{attribute 'hide_all_locals'}
FUNCTION_BLOCK FB_1_ROB EXTENDS FB_0_Base 
// IMPLEMENTS ITF_1_Robot

VAR_INPUT
	SET_R: stSettings_Rob;
	PM: FB_PointManager;
	COMM: POINTER TO FB_1_COMM := ADR(emptyCOMM);

END_VAR


VAR_OUTPUT
	HMI_ROB: stHMI_ROB;

	nCommandID: UINT;
	eCommandStatus: eProgress;
	eCommandResult: eResult := NONE;
	
	TCPPos_PLCUnit : ST_Pose;				// mm/rad
	JointPos_PLCUnit: stJoint6;			//rad
	JointVel_PLCUnit: stJoint6;
    TCPVel_PLCUnit : ST_Pose;
END_VAR

VAR
    T_W_B      : ST_TransformMatrix;		//Set in fb_Init
	index: INT;
	
	//BAHANDLER
	Idcounter: UINT:=1000;


	
	_INIT_ROB: BOOL;
	_Homed: BOOL;
  _cancelRequestID : UINT;
  _cancelNotificationSent : BOOL;
  _lifecycleStopRequested : BOOL;
  _lifecycleStopComplete : BOOL;
END_VAR

{warning 'Add property implementation'}
PROPERTY ActualJointPosition : stJoint6
GET
ActualJointPosition := JointPos_PLCUnit;
END_GET
SET
JointPos_PLCUnit:= ActualJointPosition;
END_SET
END_PROPERTY

{warning 'Add property implementation'}
  PROPERTY ActualJointVelocity : stJoint6
GET
ActualJointVelocity := JointVel_PLCUnit;
END_GET
SET
JointVel_PLCUnit := ActualJointVelocity;
END_SET
END_PROPERTY

{warning 'Add property implementation'}
  PROPERTY ActualPosition : ST_Pose
GET
ActualPosition := TCPPos_PLCUnit;
END_GET
SET
TCPPos_PLCUnit:= ActualPosition;
END_SET
END_PROPERTY

{warning 'Add property implementation'}
 PROPERTY ActualVelocity : ST_Pose
GET
ActualVelocity := TCPVel_PLCUnit;
END_GET
SET
TCPVel_PLCUnit:= ActualVelocity;
END_SET
END_PROPERTY

METHOD PROTECTED AllocateCommandID : UINT
IF Idcounter >= 65534 THEN
  Idcounter := 1001;
ELSE
	Idcounter := Idcounter + 1;
END_IF

AllocateCommandID := Idcounter;
END_METHOD

PROPERTY CanAcceptCommand : BOOL
GET
CanAcceptCommand :=
    (State = eState.Active)
    AND NOT RecoveryPending
    AND NOT ((nCommandID <> 0)
      AND ((eCommandStatus = INIT)
        OR (eCommandStatus = ACKNOWLEDGE)
        OR (eCommandStatus = RUNNING)));

IF CanAcceptCommand AND (COMM <> 0) AND (COMM <> ADR(emptyCOMM)) THEN
    CanAcceptCommand := COMM^.CanAcceptCommand;
END_IF
END_GET
END_PROPERTY

{warning 'Override with your own Method in final FB'}
METHOD CommandHandler : UINT
VAR_INPUT
    Cmd      : eCommands;
    Settings : stCommand_Settings := SETUP.emptySettings;
END_VAR

VAR

	CancelRes: BOOL;
END_VAR
(* Base implementation: unsupported. Final robot FB overrides this method. *)
CommandHandler := 0;
END_METHOD

PROPERTY CommandID : UINT
GET
CommandID := nCommandID;
END_GET
SET
 nCommandID := CommandID;
END_SET
END_PROPERTY

PROPERTY CommandResult : eResult
GET
CommandResult := COMM^.CommandResult;
END_GET
SET
eCommandResult := CommandResult;
IF (COMM <> 0) AND (COMM <> ADR(emptyCOMM)) THEN
    COMM^.CommandResult := CommandResult;
END_IF
END_SET
END_PROPERTY

PROPERTY CommandState : eProgress
GET
CommandState := COMM^.CommandState;
END_GET
SET
eCommandStatus := CommandState;
IF (COMM <> 0) AND (COMM <> ADR(emptyCOMM)) THEN
    COMM^.CommandState := CommandState;
END_IF
END_SET
END_PROPERTY

ACTION CYCLIC_ROB:
IF NOT _INIT_ROB THEN
	_INIT_ROB:=TRUE;
	SETUP_ROB();
END_IF

CYCLIC_BASE();
PM.HMI_PM.xCurrentTcp := ActualPosition;
PM(pRobot := THIS);

IF (State <> eState.Deactivating)
   AND (State <> eState.ErrorProcessing)
   AND (State <> eState.ShuttingDown) THEN
  _lifecycleStopRequested := FALSE;
  _lifecycleStopComplete := FALSE;
END_IF


// HMI display mirrors: _tcppos/_jointpos stay in PLC standard (mm/rad); display in mm/deg.
HMI_ROB.TCPPos_HMIUnit := ChangePoseToHMIStandard(Pose := TCPPos_PLCUnit);

HMI_ROB.JointPos_HMIUnit.joint1 := ChangeRealToHMIStandard(
    Value := JointPos_PLCUnit.joint1, Category := eUnitCategory.Joint);
HMI_ROB.JointPos_HMIUnit.joint2 := ChangeRealToHMIStandard(
    Value := JointPos_PLCUnit.joint2, Category := eUnitCategory.Joint);
HMI_ROB.JointPos_HMIUnit.joint3 := ChangeRealToHMIStandard(
    Value := JointPos_PLCUnit.joint3, Category := eUnitCategory.Joint);
HMI_ROB.JointPos_HMIUnit.joint4 := ChangeRealToHMIStandard(
    Value := JointPos_PLCUnit.joint4, Category := eUnitCategory.Joint);
HMI_ROB.JointPos_HMIUnit.joint5 := ChangeRealToHMIStandard(
    Value := JointPos_PLCUnit.joint5, Category := eUnitCategory.Joint);
HMI_ROB.JointPos_HMIUnit.joint6 := ChangeRealToHMIStandard(
    Value := JointPos_PLCUnit.joint6, Category := eUnitCategory.Joint);

// Adopt communication faults + health so the robot reflects its comm child.
IF COMM <> 0 AND COMM <> ADR(emptyCOMM) THEN
  COMM^.MESSENGER.ParentMessenger := ADR(MESSENGER);
	IF COMM^.State = eState.ErrorProcessing OR COMM^.MESSENGER.HasActivError THEN
        SetRecoveryMode(Mode := COMM^.RecoveryMode);
		Messenger.AddError(eMessageCategories.ParentFailed,Path,'Communication module in error');
	END_IF
END_IF




FOR index := TO_INT(LOWER_BOUND(Skills, 1)) TO TO_INT(UPPER_BOUND(Skills, 1)) DO
    IF Skills[index] <> 0 THEN
        Skills[index]^.CYCLIC_SKILL();
    END_IF
END_FOR






// --------------PROPS------------

//ActualJointPosition: DONE
//ActualJointVelocity DONE
//ActualTCPPosition: DONE
//ActualTCPVelocity: DONE
//InCollision: depend on Robot Type //TODO
//Mode: depend on RobotType	//TODO

//RobotMoving:
HMI_ROB.bMoving :=
  (ABS(TCPVel_PLCUnit.X)  > SET_R.LinearStandStillLimit) OR
  (ABS(TCPVel_PLCUnit.Y)  > SET_R.LinearStandStillLimit) OR
  (ABS(TCPVel_PLCUnit.Z)  > SET_R.LinearStandStillLimit) OR
  (ABS(TCPVel_PLCUnit.roll) > SET_R.AngularStandStillLimit) OR
  (ABS(TCPVel_PLCUnit.pitch) > SET_R.AngularStandStillLimit) OR
  (ABS(TCPVel_PLCUnit.yaw) > SET_R.AngularStandStillLimit);
	
// Generic robot command contributes to FB_0_Base.Busy. Terminal command values remain latched,
// therefore only non-terminal phases make the robot busy.
HMI_BASE.bBusy := (nCommandID <> 0)
  AND ((eCommandStatus = INIT)
    OR (eCommandStatus = ACKNOWLEDGE)
    OR (eCommandStatus = RUNNING));

IF (COMM <> 0) AND (COMM <> ADR(emptyCOMM)) THEN
  HMI_BASE.bBusy := HMI_BASE.bBusy OR COMM^.StopPending;
END_IF

// Ready means: the robot can accept a NEW semantic command now.
HMI_ROB.bOperational := Operational;
END_ACTION

METHOD PROTECTED EnsureMotionStopped : BOOL
EnsureMotionStopped := FALSE;

    IF (COMM = 0) OR (COMM = ADR(emptyCOMM)) THEN
      EnsureMotionStopped := TRUE;
      RETURN;
    END_IF

    IF NOT _lifecycleStopRequested THEN
      IF NOT COMM^.StopMotion() THEN
        Messenger.AddError(
          eMessageCategories.HardwareFailure,
          CONCAT(Path, '.StopMotion'),
          'Communication adapter rejected the lifecycle stop request');
        RETURN;
      END_IF
      _lifecycleStopRequested := TRUE;
    END_IF

    IF COMM^.MotionStopped THEN
      _lifecycleStopComplete := TRUE;
    END_IF

    EnsureMotionStopped := _lifecycleStopComplete;
END_METHOD

METHOD FB_Init : BOOL
  VAR_INPUT
    bInitRetains : BOOL;
    bInCopyCode : BOOL;
  END_VAR
  VAR
    iRobot : UINT;
  END_VAR
SUPER^.FB_Init(bInitRetains := bInitRetains, bInCopyCode := bInCopyCode);


T_W_B := FromPose(SET_R.InstallationPose);





IF SETUP.nRobCount < SETUP.MaxNrofRobots THEN
	SETUP.nRobCount := SETUP.nRobCount + 1;
	SETUP.apRobot[SETUP.nRobCount+1] := THIS;
	FB_Init := TRUE;
END_IF
END_METHOD

PROPERTY Homed : BOOL
GET
Homed:=_Homed;
END_GET
SET
_Homed:=Homed;
END_SET
END_PROPERTY

{warning 'Add method implementation '}
METHOD Homing : UINT


VAR
	Config: stCommand_Settings;
END_VAR

Config.Velocity := SET_R.HomingVelocity;

Homing:= CommandHandler(Cmd:=eCommands.Homing,Settings:=Config);
END_METHOD

PROPERTY InSavePosition : BOOL
GET
VAR
    joints : stJoint6;
END_VAR
joints := ActualJointPosition;

InSavePosition :=
    (ABS(joints.joint1 - SET_R.ManualSecurePosition.joint1) <= SET_R.SafePositionTolerance) AND
    (ABS(joints.joint2 - SET_R.ManualSecurePosition.joint2) <= SET_R.SafePositionTolerance) AND
    (ABS(joints.joint3 - SET_R.ManualSecurePosition.joint3) <= SET_R.SafePositionTolerance) AND
    (ABS(joints.joint4 - SET_R.ManualSecurePosition.joint4) <= SET_R.SafePositionTolerance) AND
    (ABS(joints.joint5 - SET_R.ManualSecurePosition.joint5) <= SET_R.SafePositionTolerance) AND
    (ABS(joints.joint6 - SET_R.ManualSecurePosition.joint6) <= SET_R.SafePositionTolerance);
END_GET
END_PROPERTY

{warning 'OVERRIDE'}
PROPERTY IsInCollision : BOOL
GET
IsInCollision := HMI_ROB.bInCollision;
END_GET
END_PROPERTY

PROPERTY IsMoving : BOOL
GET
IsMoving := HMI_ROB.bMoving;
END_GET
SET
HMI_ROB.bMoving := IsMoving;
END_SET
END_PROPERTY

METHOD MoveToHomePosition : UINT

VAR
    settings : stCommand_Settings;
END_VAR
MoveToHomePosition := 0;
settings.Velocity := SET_R.HomingVelocity;

IF PM.Load(SET_R.NameOfHomePosition) = SUCCESS THEN
    settings.Pose := PM.LoadedPose;
    MoveToHomePosition := CommandHandler(Cmd := eCommands.MoveJ, Settings := settings);
ELSE
    Messenger.AddError(eMessageCategories.MissingData, Path, 'Home Position not found, aborted');
END_IF
END_METHOD

METHOD MoveToSafePosition : UINT

VAR
    settings : stCommand_Settings;
END_VAR
settings.Velocity := SET_R.HomingVelocity;

IF SET_R.UseSavedSecurePosition THEN							//Not made: Able to save a Saveposition		
	IF PM.Load(SET_R.NameOfSavedSecurePosition) = SUCCESS THEN												
		settings.Pose := PM.LoadedPose;
		MoveToSafePosition := CommandHandler(Cmd := eCommands.MoveJ, Settings := settings);
		RETURN;
	ELSE
		Messenger.AddWarn(eMessageCategories.MissingData,Path,'Secure Position not found, using Manual Position');
		
	END_IF
END_IF


settings.Joints := SET_R.ManualSecurePosition;
MoveToSafePosition := CommandHandler(Cmd := eCommands.MoveJJoints, Settings := settings);
END_METHOD

METHOD PROTECTED OnActivate : eResult
VAR_INPUT
END_VAR

VAR
	eParentResult: eResult;
	myResult: ERESULT;
END_VAR

VAR //YOUR CODE
	succ : BOOL;
END_VAR
eParentResult := SUPER^.OnActivate();
//--------------------------------------------------
myResult:=NONE;
// ----- YOUR CODE HERE (incl. Alarms) -------------

IF Comm^.LastTransitionType = eTransitions.Activate THEN
	IF Comm^.LastTransitionResult = SUCCESS THEN
		myResult:=SUCCESS;
	END_IF
ELSE
	COMM^.Activate();
END_IF

IF SIMMODE THEN
		myResult:=SUCCESS;
END_IF

// ----- END YOUR CODE -----------------------------
//--------------------------------------------------
OnActivate := CombineResults(eParentResult,myResult);
END_METHOD

METHOD PROTECTED OnCleanup : eResult
VAR_INPUT
END_VAR

VAR
	eParentResult: eResult;
	myResult: ERESULT;
END_VAR

VAR //YOUR CODE
	succ : BOOL;
END_VAR
eParentResult := SUPER^.OnCleanup();
//--------------------------------------------------
myResult:=NONE;
// ----- YOUR CODE HERE (incl. Alarms) -------------

IF Comm^.LastTransitionType = eTransitions.Cleanup THEN
	IF Comm^.LastTransitionResult = SUCCESS THEN
		myResult:=SUCCESS;
	END_IF
ELSE
	COMM^.Cleanup();
END_IF

// ----- END YOUR CODE -----------------------------
//--------------------------------------------------
OnCleanup := CombineResults(eParentResult,myResult);
END_METHOD

METHOD PROTECTED OnConfigure : eResult
VAR_INPUT
END_VAR

VAR
	eParentResult: eResult;
	myResult: ERESULT;
END_VAR

VAR //YOUR CODE
	succ : BOOL;
END_VAR
eParentResult := SUPER^.OnConfigure();
//--------------------------------------------------
myResult:=NONE;
// ----- YOUR CODE HERE (incl. Alarms) -------------


IF Comm^.LastTransitionType = eTransitions.Configure THEN
	
	IF Comm^.LastTransitionResult = SUCCESS AND COMM^.Connected  THEN
		myResult:=SUCCESS;
	END_IF
ELSE
	COMM^.Configure();
END_IF

IF SIMMODE THEN
		myResult:=SUCCESS;
END_IF



IF NOT PM.Initialise(sName := Name) = SUCCESS THEN
	myResult:=NONE;
END_IF

PM.LoadAllFromFile();

// ----- END YOUR CODE -----------------------------
//--------------------------------------------------
OnConfigure := CombineResults(eParentResult,myResult);
END_METHOD

METHOD PROTECTED OnDeactivate : eResult
VAR_INPUT
END_VAR

VAR
	eParentResult: eResult;
	myResult: ERESULT;
END_VAR

VAR //YOUR CODE
	succ : BOOL;
END_VAR
eParentResult := SUPER^.OnDeactivate();

IF NOT EnsureMotionStopped() THEN
  OnDeactivate := CombineResults(eParentResult, eResult.NONE);
  RETURN;
END_IF
//--------------------------------------------------
myResult:=NONE;
// ----- YOUR CODE HERE (incl. Alarms) -------------

IF Comm^.LastTransitionType = eTransitions.Deactivate THEN
	IF Comm^.LastTransitionResult = SUCCESS THEN
		myResult:=SUCCESS;
	END_IF
ELSE
	COMM^.Deactivate();
END_IF

// ----- END YOUR CODE -----------------------------
//--------------------------------------------------
OnDeactivate := CombineResults(eParentResult,myResult);
END_METHOD

METHOD PROTECTED OnError : eResult
VAR_INPUT
END_VAR

VAR
	eParentResult: eResult;
	myResult: ERESULT;
END_VAR

VAR //YOUR CODE
	succ : BOOL;
END_VAR
eParentResult := SUPER^.OnError();
myResult := NONE;

IF NOT EnsureMotionStopped() THEN
  OnError := CombineResults(eParentResult, eResult.NONE);
  RETURN;
END_IF

// Communication recovery owns its own policy. The robot only waits for it and
// propagates a more restrictive recovery mode upward.
IF (COMM = 0) OR (COMM = ADR(emptyCOMM)) THEN
    myResult := SUCCESS;
ELSIF COMM^.State = eState.ErrorProcessing THEN
    SetRecoveryMode(Mode := COMM^.RecoveryMode);
    myResult := NONE;
ELSIF COMM^.MESSENGER.HasActivError THEN
    SetRecoveryMode(Mode := COMM^.RecoveryMode);
    myResult := NONE;
ELSE
    myResult := SUCCESS;
END_IF

OnError := CombineResults(eParentResult, myResult);
END_METHOD

METHOD PROTECTED OnShutdown : eResult
VAR_INPUT
END_VAR

VAR
	eParentResult: eResult;
	myResult: ERESULT;
END_VAR

VAR //YOUR CODE
	succ : BOOL;
END_VAR
eParentResult := SUPER^.OnShutdown();

IF NOT EnsureMotionStopped() THEN
  OnShutdown := CombineResults(eParentResult, eResult.NONE);
  RETURN;
END_IF
//--------------------------------------------------
myResult:=NONE;
// ----- YOUR CODE HERE (incl. Alarms) -------------

IF Comm^.LastTransitionType = eTransitions.Shutdown THEN
	IF Comm^.LastTransitionResult = SUCCESS THEN
		myResult:=SUCCESS;
	END_IF
ELSE
	COMM^.Shutdown();
END_IF

// ----- END YOUR CODE -----------------------------
//--------------------------------------------------
OnShutdown := CombineResults(eParentResult,myResult);
END_METHOD

PROPERTY Operational : BOOL
SET
SUPER^.Operational := Operational AND COMM^.Operational;
END_SET
END_PROPERTY

PROPERTY Powered : BOOL
GET
Powered:=HMI_ROB.bPowered;
END_GET
SET
HMI_ROB.bPowered:=Powered;
END_SET
END_PROPERTY

{attribute 'TcRpcEnable':='1'}
METHOD PUBLIC Reset : eResult
VAR_INPUT
END_VAR
Reset := SUPER^.Reset();

// A robot acknowledgement is propagated only to a communication child that is
// itself waiting in ErrorProcessing. It is still only permission to recover.
IF (COMM <> 0) AND (COMM <> ADR(emptyCOMM)) AND (COMM^.State = eState.ErrorProcessing) THEN
    COMM^.Reset();
END_IF
END_METHOD

METHOD PUBLIC ResolveAbsoluteTarget : BOOL
VAR_INPUT
    TargetIn : ST_Pose;
    Frame    : eRefFrame;

    // Transformation of robot BRF expressed in WRF
    T_W_B    : ST_TransformMatrix;

    // Custom user frame expressed in BRF (only used for eRefFrame.CRF).
    T_B_Custom : ST_TransformMatrix;
END_VAR

VAR_OUTPUT
    Target : ST_Pose;
END_VAR

VAR
    T_W_Target : ST_TransformMatrix;
    T_B_Target : ST_TransformMatrix;
    T_B_W      : ST_TransformMatrix;
    T_C_Target : ST_TransformMatrix;
END_VAR
ResolveAbsoluteTarget := FALSE;


//--------------------------------------------------
// Resolve absolute Cartesian target into BRF.
// Output is ALWAYS in PLC standard units (m, rad).
//--------------------------------------------------

CASE Frame OF


    eRefFrame.BRF:

        Target := TargetIn;


    eRefFrame.WRF:

        // T_B_Target = inv(T_W_B) * T_W_Target
        T_W_Target := FromPose(Pose := TargetIn);
        T_B_W := Inverse(T := T_W_B);
        T_B_Target := Multiply(A := T_B_W, B := T_W_Target);
        Target := ToPose(T := T_B_Target);


//     eRefFrame.CRF:
// 
//         // Target expressed in custom frame; T_B_Custom is that frame in BRF.
//         // T_B_Target = T_B_Custom * T_C_Target
//         T_C_Target := FromPose(Pose := TargetIn);
//         T_B_Target := Multiply(A := T_B_Custom, B := T_C_Target);
//         Target := ToPose(T := T_B_Target);


    eRefFrame.TRF:

        // Absolute TRF is intentionally undefined; use ResolveRelativeTarget instead.
        RETURN;


    ELSE

        RETURN;

END_CASE


ResolveAbsoluteTarget := TRUE;
END_METHOD

METHOD PUBLIC ResolveRelativeTarget : BOOL
VAR_INPUT
    Delta      : ST_Pose;		//Offset expressed in the selected Frame
    Frame      : eRefFrame;

   
//     T_B_Custom : ST_TransformMatrix;  // Custom user frame expressed in BRF (only used for eRefFrame.CRF).
END_VAR

VAR_OUTPUT
    Target : ST_Pose;
END_VAR

VAR
    TCurrent    : ST_TransformMatrix;
    TDelta      : ST_TransformMatrix;
    TResult     : ST_TransformMatrix;

    T_W_Current : ST_TransformMatrix;
    T_W_Target  : ST_TransformMatrix;
    T_B_W       : ST_TransformMatrix;

    T_C_B       : ST_TransformMatrix;
    T_C_Current : ST_TransformMatrix;
    T_C_Target  : ST_TransformMatrix;
END_VAR
ResolveRelativeTarget := FALSE;


// CurrentTCP is always expected in BRF (PLC standard units).
TCurrent := FromPose(Pose := ActualPosition);
TDelta   := FromPose(Pose := Delta);


CASE Frame OF


    eRefFrame.BRF:

        // T_B_Target = T_B_Delta * T_B_Current
        TResult := Multiply(A := TDelta, B := TCurrent);


    eRefFrame.WRF:

        // T_W_Current = T_W_B * T_B_Current
        T_W_Current := Multiply(A := T_W_B, B := TCurrent);

        // T_W_Target = T_W_Delta * T_W_Current
        T_W_Target := Multiply(A := TDelta, B := T_W_Current);

        // T_B_Target = inv(T_W_B) * T_W_Target
        T_B_W := Inverse(T := T_W_B);
        TResult := Multiply(A := T_B_W, B := T_W_Target);


    eRefFrame.TRF:

        // Delta in current tool frame: T_B_Target = T_B_Current * T_T_Delta
        TResult := Multiply(A := TCurrent, B := TDelta);

// 
//     eRefFrame.CRF:
// 
//         // Delta expressed in a custom frame given by T_B_Custom.
//         // T_C_Current = inv(T_B_Custom) * T_B_Current
//         // T_C_Target  = T_C_Delta * T_C_Current
//         // T_B_Target  = T_B_Custom * T_C_Target
//         T_C_B := Inverse(T := T_B_Custom);
//         T_C_Current := Multiply(A := T_C_B, B := TCurrent);
//         T_C_Target  := Multiply(A := TDelta, B := T_C_Current);
//         TResult := Multiply(A := T_B_Custom, B := T_C_Target);
// 

    ELSE

        RETURN;

END_CASE


// Result is ALWAYS expressed in BRF, in PLC standard units.
Target := ToPose(T := TResult);


ResolveRelativeTarget := TRUE;
END_METHOD

ACTION SETUP_ROB:
FOR j:= TO_INT(LOWER_BOUND(Skills, 1)) TO TO_INT(UPPER_BOUND(Skills, 1)) DO //fb_init??
	IF Skills[j]<>0 THEN
		Skills[j]^.pOwner:=THIS;
	END_IF
	
	SUPER^.SET_B:=SET_R;
END_FOR

PM.NameOfRobot:=Name;
PM.MESSENGER.ParentMessenger:=ADR(Messenger);
END_ACTION

PROPERTY SpeedOverride : REAL
GET
SpeedOverride := HMI_ROB.ValueOfSpeedOverride;
END_GET
SET
IF (SpeedOverride < 0.001) OR (SpeedOverride > 100.0) THEN
    HMI_ROB.ValueOfSpeedOverride := 100; 
ELSE
	HMI_ROB.ValueOfSpeedOverride := SpeedOverride;
END_IF
END_SET
END_PROPERTY

METHOD PUBLIC StopMotion : BOOL
StopMotion := FALSE;
IF (COMM <> 0) AND (COMM <> ADR(emptyCOMM)) THEN
    StopMotion := COMM^.StopMotion();
END_IF
END_METHOD

END_FUNCTION_BLOCK

(* stored: Version 1.1.0.1, ProductVersion 3.1.4026.18
   POU FB_1_ROB: Id {7ce28b50-28f8-4d4c-bb25-1006bf064637}, SpecialFunc None
   Folder Command: Id {dbd57985-4d16-4bc8-859d-d7e9147003e9}
   Folder Generic Control: Id {d269719e-4481-455b-8abd-a0a346547cd3}
   Folder Generic Status: Id {c1e8e35a-1828-4d72-a2cb-3aa1cc7ab721}
   Folder StateControl: Id {306f9b72-2cb2-4dec-88a3-0a1776eb8cb9}
   Folder Transformations: Id {12df3c52-cfe6-44d7-9d03-72f041d59ebd}
   Property ActualJointPosition: Id {c68b9d82-514b-4e83-b58e-69cf77564b19}
   Get Get: Id {2b353ef5-5db5-4268-89e1-d980ddc297fa}
   Set Set: Id {5200eb36-b713-4fd9-acea-1d29264b6a02}
   Property ActualJointVelocity: Id {947a6f2a-4f8a-49d4-9aa5-6819f46128db}
   Get Get: Id {bcb260e7-58e3-43cb-b050-6f35e444f22e}
   Set Set: Id {05d019ac-6445-4c92-986d-31cfda1313fe}
   Property ActualPosition: Id {0ea3c3d9-9984-43b2-ac68-a1a8d409d11e}
   Get Get: Id {019c7e94-91db-4b36-9e6e-9be7d9fb51c3}
   Set Set: Id {44131c92-965f-457b-85c5-727220982875}
   Property ActualVelocity: Id {cd04f35a-047d-478b-8cf7-b18ee8d2a4f9}
   Get Get: Id {c88b221c-0030-413b-abf3-a401e3f71088}
   Set Set: Id {e2c2d2bc-653c-4555-bb7b-571a1ce7564a}
   Method AllocateCommandID: Id {4de8c731-a286-4ca0-9f0f-d43282496255}
   Property CanAcceptCommand: Id {ecdb9c1a-5dfb-4d8b-9dc8-7992c493eb98}
   Get Get: Id {5ce2868b-d6c9-486f-9f2d-1ce0bec46b73}
   Method CommandHandler: Id {83e2d403-4d26-4906-9c94-3843f0c8311a}
   Property CommandID: Id {d97dbde2-fb4a-4a46-80b5-95e72bfb597d}
   Get Get: Id {f42bf0bc-af24-437d-951f-342952505cbf}
   Set Set: Id {4147eece-a2c2-4265-9a5a-16d2dfe5e198}
   Property CommandResult: Id {2743123b-b65d-4f7b-9069-9ec61dd72659}
   Get Get: Id {9324d1a7-b98e-458b-8e19-2f6253d717cd}
   Set Set: Id {c29cbfae-44af-4688-9231-cff74c2ee443}
   Property CommandState: Id {6c07ca32-53d2-4833-85fe-587d61a168d6}
   Get Get: Id {f225aadd-c904-4018-87ed-75348f6fbad4}
   Set Set: Id {6eb2d0d5-717a-4e91-ab0f-27827dd25d8f}
   Action CYCLIC_ROB: Id {ebf16c89-c511-406b-9426-1ade99c4f730}
   Method EnsureMotionStopped: Id {e0f87680-a790-4af7-9869-97c5d171646e}
   Method FB_Init: Id {7b302bc2-af12-4e54-8aa2-dca07a2dd5cc}
   Property Homed: Id {0293db6b-1676-4fdb-900d-d48a6f2fe520}
   Get Get: Id {8296b06f-a6d6-4c3f-ac49-4a977d01c83b}
   Set Set: Id {9fd8795d-992d-4416-a301-e62e92d902d5}
   Method Homing: Id {332921a2-9f70-499b-943d-00519405a468}
   Property InSavePosition: Id {0b1ac6ae-f2f1-4986-8684-c6891da4f895}
   Get Get: Id {f07a4056-55e2-4a4d-b3fa-f23e3592a78e}
   Property IsInCollision: Id {8eea56b9-50ca-4510-b567-db19e3eca5c7}
   Get Get: Id {885867df-c0d3-4443-aec9-8d2b982d6c40}
   Property IsMoving: Id {35ca0c87-c7ee-4f80-a87b-f8e0bf6781ef}
   Get Get: Id {4af7c180-96b4-478d-9ba7-15a9132d033d}
   Set Set: Id {8c3ef50b-f0bb-4f67-b971-f8d926a0360c}
   Method MoveToHomePosition: Id {c14a5534-c5f9-4fac-a596-50be651bd65e}
   Method MoveToSafePosition: Id {1460c5aa-e9ef-4e0e-a2bc-5ac3c6af9cb6}
   Method OnActivate: Id {c53d2e09-95f6-4470-b92a-1736ae881f81}
   Method OnCleanup: Id {734e8874-f49e-492d-ae48-dcfbab1bde00}
   Method OnConfigure: Id {405f6b01-72da-4ba1-a9bb-82f8cc48639e}
   Method OnDeactivate: Id {0745a082-7014-41b6-ad3f-f3e98871c693}
   Method OnError: Id {241d30dc-f0b7-4588-8953-d135c03fba6b}
   Method OnShutdown: Id {b65c468a-c599-4af9-bafe-bb502871193c}
   Property Operational: Id {8f2c7f81-6dd1-4fa4-9c6b-42ea40f162a7}
   Set Set: Id {54d641e5-fe9d-4485-81ab-0a9ea2273a9e}
   Property Powered: Id {110ec326-6e7c-44f2-915c-7dafa2d7f0fb}
   Get Get: Id {9c1bf6ab-a19d-4b56-b4f0-7114872379b5}
   Set Set: Id {368defae-d77c-481a-9a3f-7c58e4d8aee0}
   Method Reset: Id {2c7d1a90-4e33-4b71-9a02-8f1a2b3c4d50}
   Method ResolveAbsoluteTarget: Id {b77bfcd9-1d5b-42ab-9650-d1a07eb2b312}
   Method ResolveRelativeTarget: Id {7316aa83-122c-4f87-a413-cdf614e4c220}
   Action SETUP_ROB: Id {a4cb3038-46c5-4081-b870-1e91e16123a5}
   Property SpeedOverride: Id {264b7b02-b2eb-4a64-8c70-3421c0dcfab6}
   Get Get: Id {bf44923c-76c4-4a55-8a7f-83936e0fb927}
   Set Set: Id {00d512c8-cfe3-49b4-ac1a-2fe68ecc1046}
   Method StopMotion: Id {2a9ef1f1-bebf-42b7-9028-b416fb72a19e} *)
